// Mitsubishi GX Developer project: 310HGV18J11Y减 改扫码181011   PLC: FX3G

PROGRAM MAIN
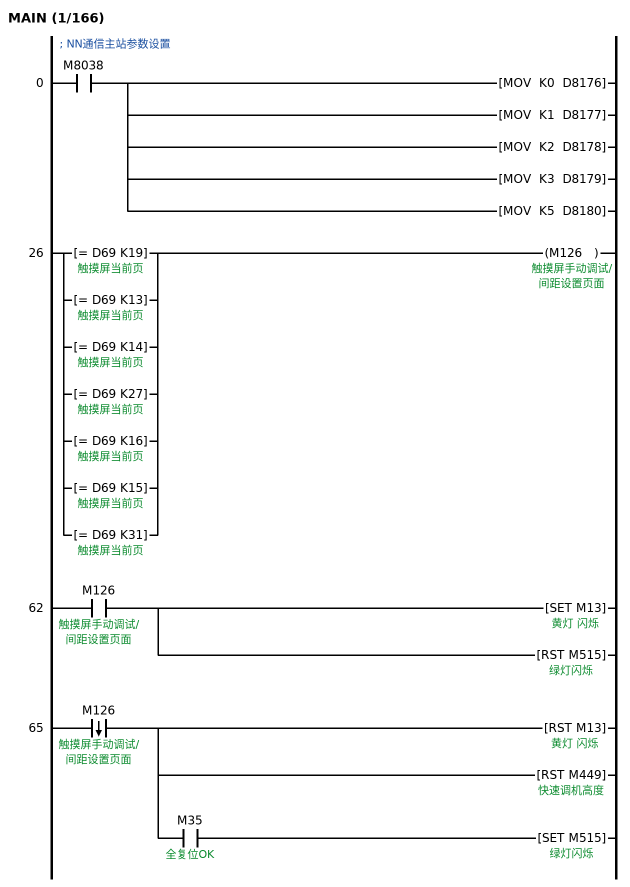
; NN通信主站参数设置
0     LD      M8038
      MOV     K0 D8176
      MOV     K1 D8177
      MOV     K2 D8178
      MOV     K3 D8179
      MOV     K5 D8180
26    LD=     D69 K19  ; 触摸屏当前页
      OR=     D69 K13  ; 触摸屏当前页
      OR=     D69 K14  ; 触摸屏当前页
      OR=     D69 K27  ; 触摸屏当前页
      OR=     D69 K16  ; 触摸屏当前页
      OR=     D69 K15  ; 触摸屏当前页
      OR=     D69 K31  ; 触摸屏当前页
      OUT     M126  ; 触摸屏手动调试/间距设置页面
62    LD      M126  ; 触摸屏手动调试/间距设置页面
      SET     M13  ; 黄灯 闪烁
      RST     M515  ; 绿灯闪烁
65    LDF     M126  ; 触摸屏手动调试/间距设置页面
      RST     M13  ; 黄灯 闪烁
      RST     M449  ; 快速调机高度
      AND     M35  ; 全复位OK
      SET     M515  ; 绿灯闪烁
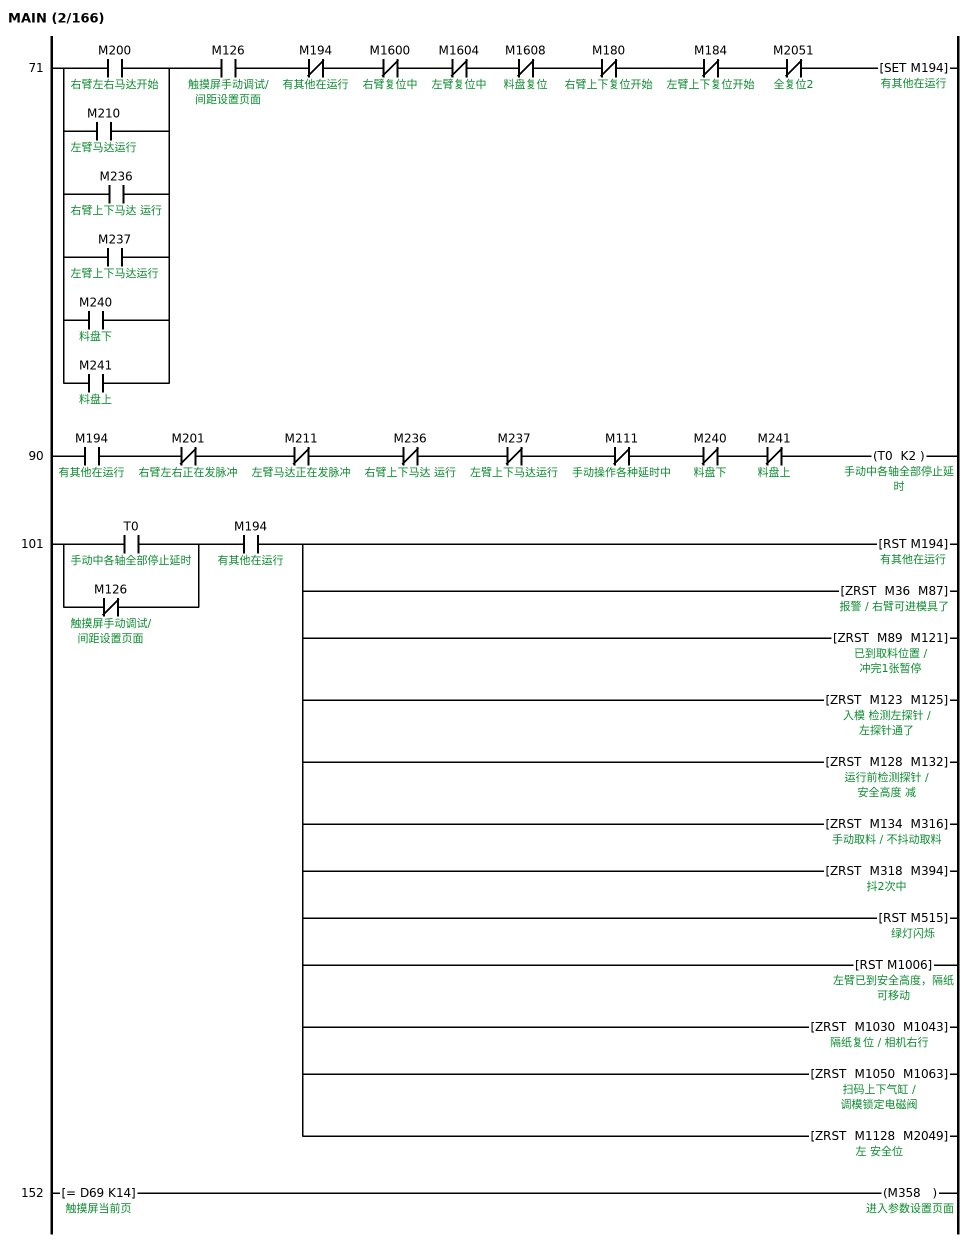
71    LD      M200  ; 右臂左右马达开始
      OR      M210  ; 左臂马达运行
      OR      M236  ; 右臂上下马达 运行
      OR      M237  ; 左臂上下马达运行
      OR      M240  ; 料盘下
      OR      M241  ; 料盘上
      AND     M126  ; 触摸屏手动调试/间距设置页面
      ANI     M194  ; 有其他在运行
      ANI     M1600  ; 右臂复位中
      ANI     M1604  ; 左臂复位中
      ANI     M1608  ; 料盘复位
      ANI     M180  ; 右臂上下复位开始
      ANI     M184  ; 左臂上下复位开始
      ANI     M2051  ; 全复位2
      SET     M194  ; 有其他在运行
90    LD      M194  ; 有其他在运行
      ANI     M201  ; 右臂左右正在发脉冲
      ANI     M211  ; 左臂马达正在发脉冲
      ANI     M236  ; 右臂上下马达 运行
      ANI     M237  ; 左臂上下马达运行
      ANI     M111  ; 手动操作各种延时中
      ANI     M240  ; 料盘下
      ANI     M241  ; 料盘上
      OUT     T0 K2  ; 手动中各轴全部停止延时
101   LD      T0  ; 手动中各轴全部停止延时
      ORI     M126  ; 触摸屏手动调试/间距设置页面
      AND     M194  ; 有其他在运行
      RST     M194  ; 有其他在运行
      ZRST    M36 M87  ; 报警 / 右臂可进模具了
      ZRST    M89 M121  ; 已到取料位置 / 冲完1张暂停
      ZRST    M123 M125  ; 入模 检测左探针 / 左探针通了
      ZRST    M128 M132  ; 运行前检测探针 / 安全高度 减
      ZRST    M134 M316  ; 手动取料 / 不抖动取料
      ZRST    M318 M394  ; 抖2次中
      RST     M515  ; 绿灯闪烁
      RST     M1006  ; 左臂已到安全高度，隔纸可移动
      ZRST    M1030 M1043  ; 隔纸复位 / 相机右行
      ZRST    M1050 M1063  ; 扫码上下气缸 / 调模锁定电磁阀
      ZRST    M1128 M2049  ; 左 安全位
152   LD=     D69 K14  ; 触摸屏当前页
      OUT     M358  ; 进入参数设置页面
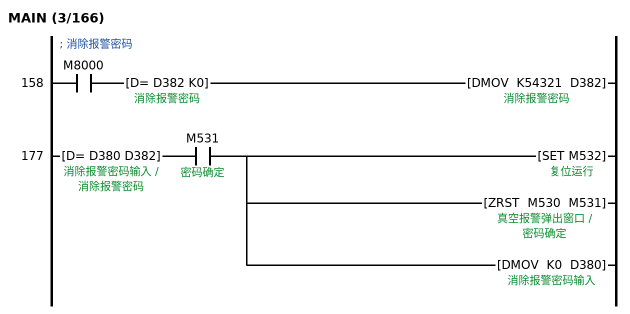
; 消除报警密码
158   LD      M8000
      ANDD=   D382 K0  ; 消除报警密码
      DMOV    K54321 D382
177   LDD=    D380 D382  ; 消除报警密码输入 / 消除报警密码
      AND     M531  ; 密码确定
      SET     M532  ; 复位运行
      ZRST    M530 M531  ; 真空报警弹出窗口
      DMOV    K0 D380
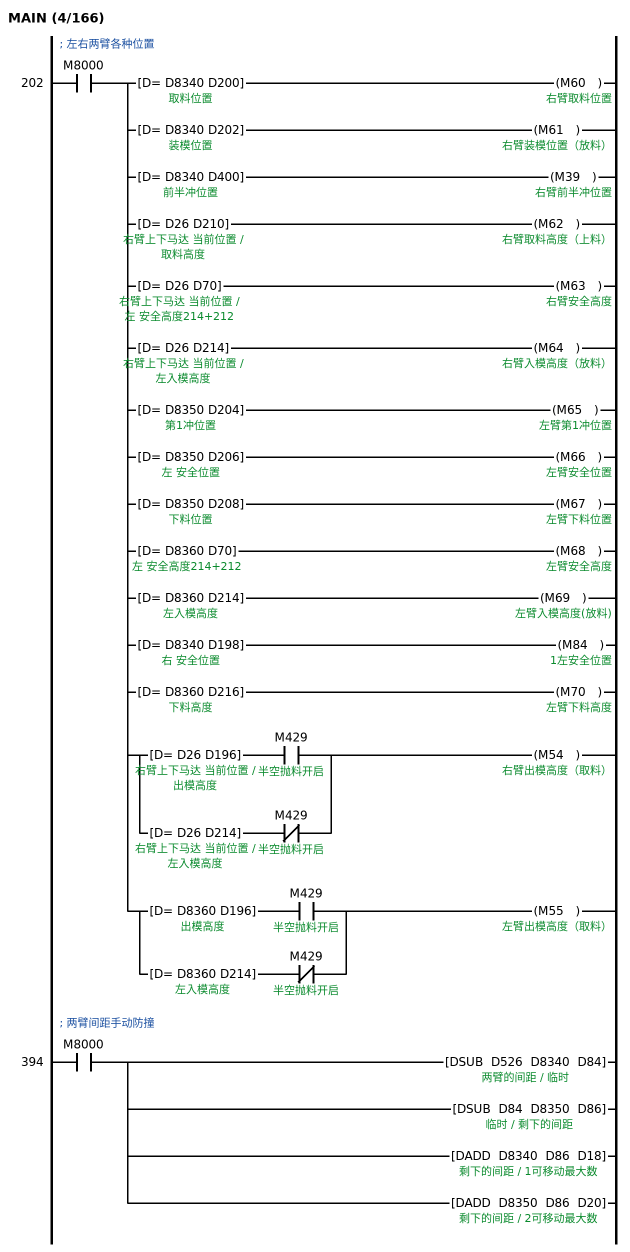
; 左右两臂各种位置
202   LD      M8000
      MPS
      ANDD=   D8340 D200  ; 取料位置
      OUT     M60  ; 右臂取料位置
      MRD
      ANDD=   D8340 D202  ; 装模位置
      OUT     M61  ; 右臂装模位置（放料）
      MRD
      ANDD=   D8340 D400  ; 前半冲位置
      OUT     M39  ; 右臂前半冲位置
      MRD
      ANDD=   D26 D210  ; 右臂上下马达 当前位置 / 取料高度
      OUT     M62  ; 右臂取料高度（上料）
      MRD
      ANDD=   D26 D70  ; 右臂上下马达 当前位置 / 左 安全高度214+212
      OUT     M63  ; 右臂安全高度
      MRD
      ANDD=   D26 D214  ; 右臂上下马达 当前位置 / 左入模高度
      OUT     M64  ; 右臂入模高度（放料）
      MRD
      ANDD=   D8350 D204  ; 第1冲位置
      OUT     M65  ; 左臂第1冲位置
      MRD
      ANDD=   D8350 D206  ; 左 安全位置
      OUT     M66  ; 左臂安全位置
      MRD
      ANDD=   D8350 D208  ; 下料位置
      OUT     M67  ; 左臂下料位置
      MRD
      ANDD=   D8360 D70  ; 左 安全高度214+212
      OUT     M68  ; 左臂安全高度
      MRD
      ANDD=   D8360 D214  ; 左入模高度
      OUT     M69  ; 左臂入模高度(放料)
      MRD
      ANDD=   D8340 D198  ; 右 安全位置
      OUT     M84  ; 1左安全位置
      MRD
      ANDD=   D8360 D216  ; 下料高度
      OUT     M70  ; 左臂下料高度
      MRD
      LDD=    D26 D196  ; 右臂上下马达 当前位置 / 出模高度
      AND     M429  ; 半空抛料开启
      LDD=    D26 D214  ; 右臂上下马达 当前位置 / 左入模高度
      ANI     M429  ; 半空抛料开启
      ORB
      ANB
      OUT     M54  ; 右臂出模高度（取料）
      MPP
      LDD=    D8360 D196  ; 出模高度
      AND     M429  ; 半空抛料开启
      LDD=    D8360 D214  ; 左入模高度
      ANI     M429  ; 半空抛料开启
      ORB
      ANB
      OUT     M55  ; 左臂出模高度（取料）
; 两臂间距手动防撞
394   LD      M8000
      DSUB    D526 D8340 D84  ; 两臂的间距 / 临时
      DSUB    D84 D8350 D86  ; 剩下的间距
      DADD    D8340 D86 D18  ; 1可移动最大数
      DADD    D8350 D86 D20  ; 2可移动最大数
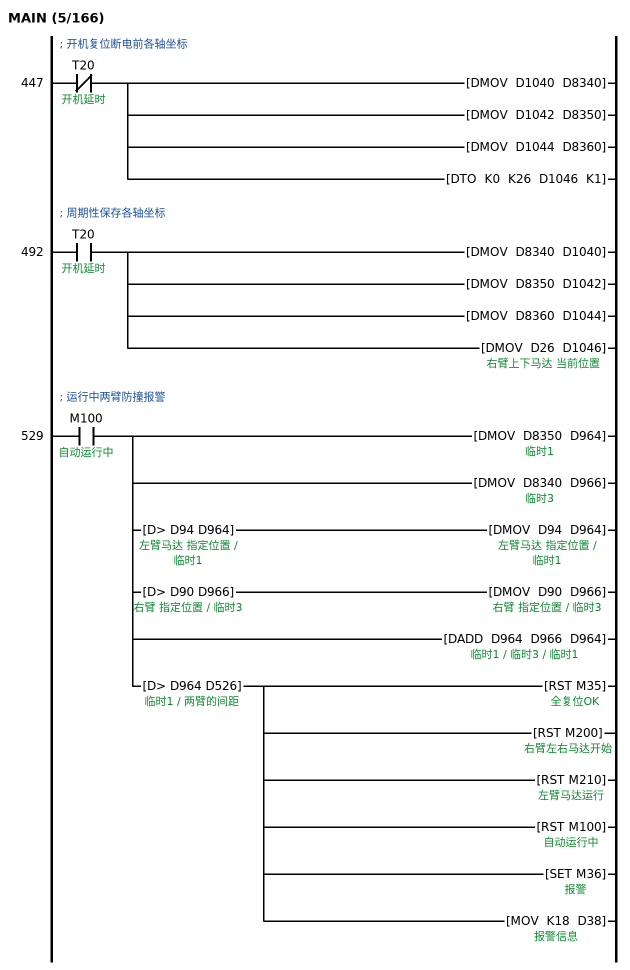
; 开机复位断电前各轴坐标
447   LDI     T20  ; 开机延时
      DMOV    D1040 D8340
      DMOV    D1042 D8350
      DMOV    D1044 D8360
      DTO     K0 K26 D1046 K1
; 周期性保存各轴坐标
492   LD      T20  ; 开机延时
      DMOV    D8340 D1040
      DMOV    D8350 D1042
      DMOV    D8360 D1044
      DMOV    D26 D1046
; 运行中两臂防撞报警
529   LD      M100  ; 自动运行中
      DMOV    D8350 D964  ; 临时1
      DMOV    D8340 D966  ; 临时3
      MPS
      ANDD>   D94 D964  ; 左臂马达 指定位置 / 临时1
      DMOV    D94 D964
      MRD
      ANDD>   D90 D966  ; 右臂 指定位置 / 临时3
      DMOV    D90 D966
      MPP
      DADD    D964 D966 D964
      ANDD>   D964 D526  ; 临时1 / 两臂的间距
      RST     M35  ; 全复位OK
      RST     M200  ; 右臂左右马达开始
      RST     M210  ; 左臂马达运行
      RST     M100  ; 自动运行中
      SET     M36  ; 报警
      MOV     K18 D38  ; 报警信息
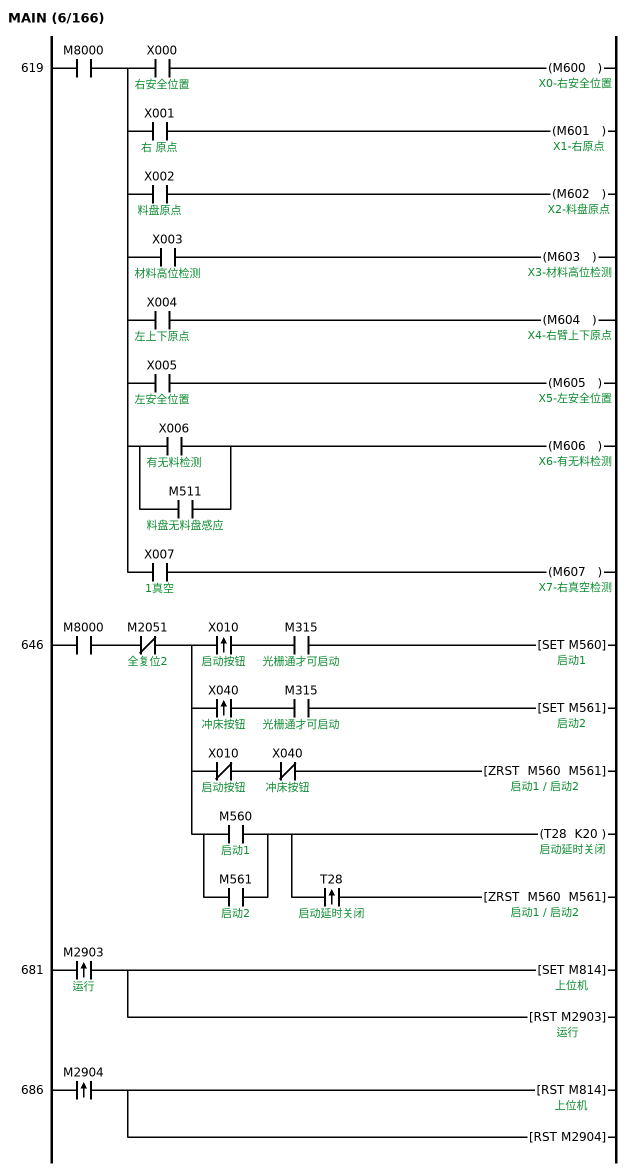
619   LD      M8000
      MPS
      AND     X000  ; 右安全位置
      OUT     M600  ; X0-右安全位置
      MRD
      AND     X001  ; 右 原点
      OUT     M601  ; X1-右原点
      MRD
      AND     X002  ; 料盘原点
      OUT     M602  ; X2-料盘原点
      MRD
      AND     X003  ; 材料高位检测
      OUT     M603  ; X3-材料高位检测
      MRD
      AND     X004  ; 左上下原点
      OUT     M604  ; X4-右臂上下原点
      MRD
      AND     X005  ; 左安全位置
      OUT     M605  ; X5-左安全位置
      MRD
      LD      X006  ; 有无料检测
      OR      M511  ; 料盘无料盘感应
      ANB
      OUT     M606  ; X6-有无料检测
      MPP
      AND     X007  ; 1真空
      OUT     M607  ; X7-右真空检测
646   LD      M8000
      ANI     M2051  ; 全复位2
      MPS
      ANDP    X010  ; 启动按钮
      AND     M315  ; 光栅通才可启动
      SET     M560  ; 启动1
      MRD
      ANDP    X040  ; 冲床按钮
      AND     M315  ; 光栅通才可启动
      SET     M561  ; 启动2
      MRD
      ANI     X010  ; 启动按钮
      ANI     X040  ; 冲床按钮
      ZRST    M560 M561
      MPP
      LD      M560  ; 启动1
      OR      M561  ; 启动2
      ANB
      OUT     T28 K20  ; 启动延时关闭
      ANDP    T28  ; 启动延时关闭
      ZRST    M560 M561
681   LDP     M2903  ; 运行
      SET     M814  ; 上位机
      RST     M2903  ; 运行
686   LDP     M2904
      RST     M814  ; 上位机
      RST     M2904
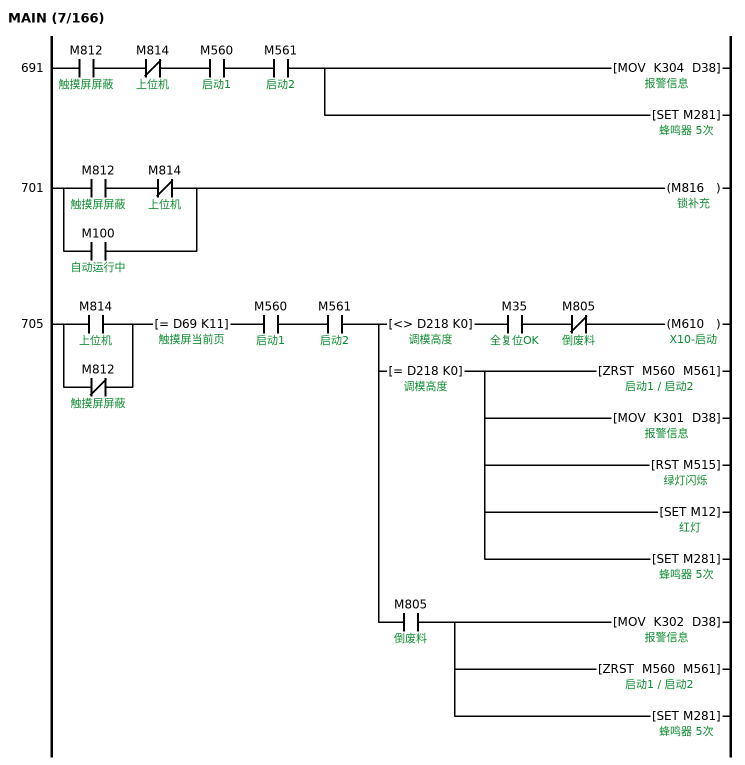
691   LD      M812  ; 触摸屏屏蔽
      ANI     M814  ; 上位机
      AND     M560  ; 启动1
      AND     M561  ; 启动2
      MOV     K304 D38
      SET     M281  ; 蜂鸣器 5次
701   LD      M812  ; 触摸屏屏蔽
      ANI     M814  ; 上位机
      OR      M100  ; 自动运行中
      OUT     M816  ; 锁补充
705   LD      M814  ; 上位机
      ORI     M812  ; 触摸屏屏蔽
      AND=    D69 K11  ; 触摸屏当前页
      AND     M560  ; 启动1
      AND     M561  ; 启动2
      MPS
      AND<>   D218 K0  ; 调模高度
      AND     M35  ; 全复位OK
      ANI     M805  ; 倒废料
      OUT     M610  ; X10-启动
      MRD
      AND=    D218 K0  ; 调模高度
      ZRST    M560 M561
      MOV     K301 D38
      RST     M515  ; 绿灯闪烁
      SET     M12  ; 红灯
      SET     M281  ; 蜂鸣器 5次
      MPP
      AND     M805  ; 倒废料
      MOV     K302 D38
      ZRST    M560 M561
      SET     M281  ; 蜂鸣器 5次
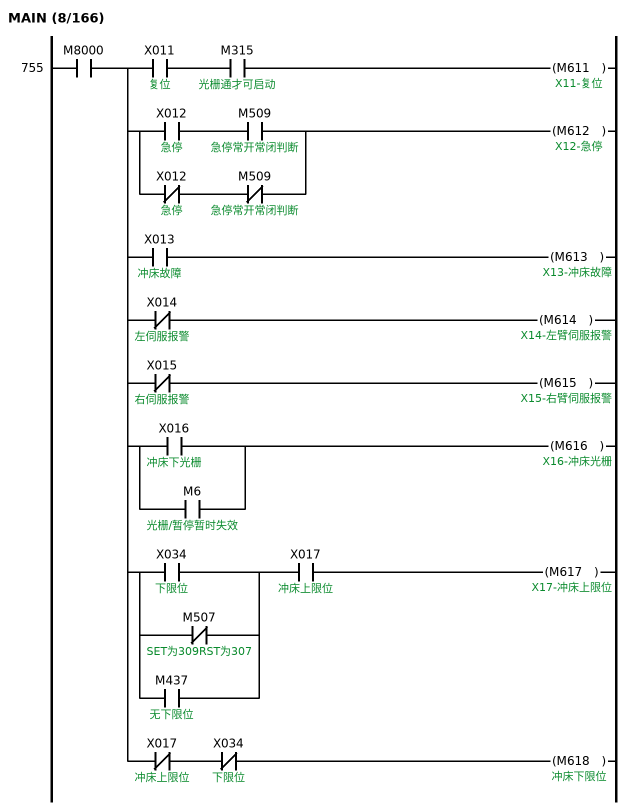
755   LD      M8000
      MPS
      AND     X011  ; 复位
      AND     M315  ; 光栅通才可启动
      OUT     M611  ; X11-复位
      MRD
      LD      X012  ; 急停
      AND     M509  ; 急停常开常闭判断
      LDI     X012  ; 急停
      ANI     M509  ; 急停常开常闭判断
      ORB
      ANB
      OUT     M612  ; X12-急停
      MRD
      AND     X013  ; 冲床故障
      OUT     M613  ; X13-冲床故障
      MRD
      ANI     X014  ; 左伺服报警
      OUT     M614  ; X14-左臂伺服报警
      MRD
      ANI     X015  ; 右伺服报警
      OUT     M615  ; X15-右臂伺服报警
      MRD
      LD      X016  ; 冲床下光栅
      OR      M6  ; 光栅/暂停暂时失效
      ANB
      OUT     M616  ; X16-冲床光栅
      MRD
      LD      X034  ; 下限位
      ORI     M507  ; SET为309RST为307
      OR      M437  ; 无下限位
      ANB
      AND     X017  ; 冲床上限位
      OUT     M617  ; X17-冲床上限位
      MPP
      ANI     X017  ; 冲床上限位
      ANI     X034  ; 下限位
      OUT     M618  ; 冲床下限位
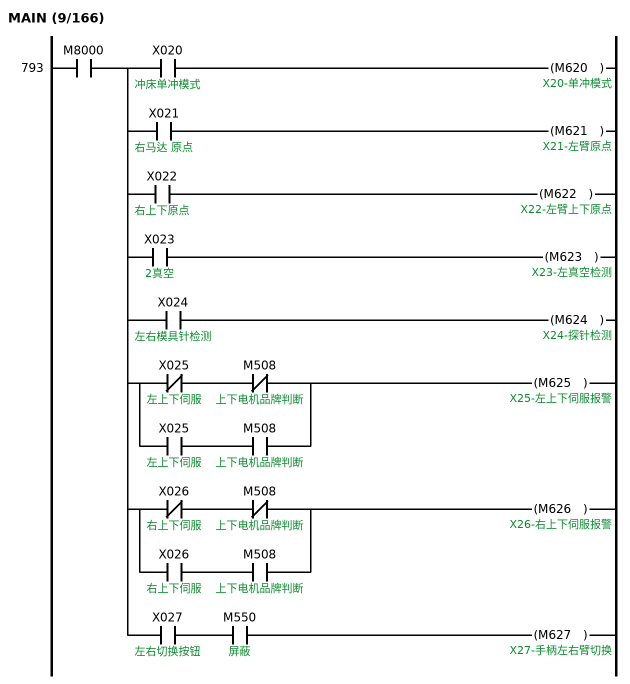
793   LD      M8000
      MPS
      AND     X020  ; 冲床单冲模式
      OUT     M620  ; X20-单冲模式
      MRD
      AND     X021  ; 右马达 原点
      OUT     M621  ; X21-左臂原点
      MRD
      AND     X022  ; 右上下原点
      OUT     M622  ; X22-左臂上下原点
      MRD
      AND     X023  ; 2真空
      OUT     M623  ; X23-左真空检测
      MRD
      AND     X024  ; 左右模具针检测
      OUT     M624  ; X24-探针检测
      MRD
      LDI     X025  ; 左上下伺服
      ANI     M508  ; 上下电机品牌判断
      LD      X025  ; 左上下伺服
      AND     M508  ; 上下电机品牌判断
      ORB
      ANB
      OUT     M625  ; X25-左上下伺服报警
      MRD
      LDI     X026  ; 右上下伺服
      ANI     M508  ; 上下电机品牌判断
      LD      X026  ; 右上下伺服
      AND     M508  ; 上下电机品牌判断
      ORB
      ANB
      OUT     M626  ; X26-右上下伺服报警
      MPP
      AND     X027  ; 左右切换按钮
      AND     M550  ; 屏蔽
      OUT     M627  ; X27-手柄左右臂切换
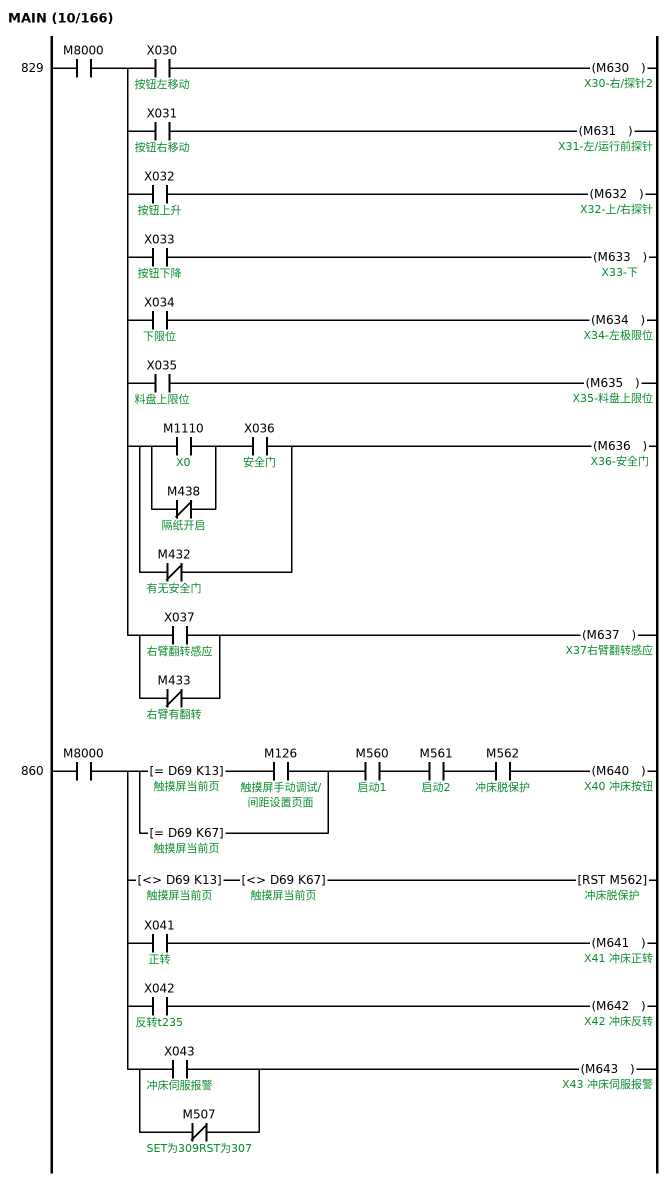
829   LD      M8000
      MPS
      AND     X030  ; 按钮左移动
      OUT     M630  ; X30-右/探针2
      MRD
      AND     X031  ; 按钮右移动
      OUT     M631  ; X31-左/运行前探针
      MRD
      AND     X032  ; 按钮上升
      OUT     M632  ; X32-上/右探针
      MRD
      AND     X033  ; 按钮下降
      OUT     M633  ; X33-下
      MRD
      AND     X034  ; 下限位
      OUT     M634  ; X34-左极限位
      MRD
      AND     X035  ; 料盘上限位
      OUT     M635  ; X35-料盘上限位
      MRD
      LD      M1110  ; X0
      ORI     M438  ; 隔纸开启
      AND     X036  ; 安全门
      ORI     M432  ; 有无安全门
      ANB
      OUT     M636  ; X36-安全门
      MPP
      LD      X037  ; 右臂翻转感应
      ORI     M433  ; 右臂有翻转
      ANB
      OUT     M637  ; X37右臂翻转感应
860   LD      M8000
      MPS
      LD=     D69 K13  ; 触摸屏当前页
      AND     M126  ; 触摸屏手动调试/间距设置页面
      OR=     D69 K67  ; 触摸屏当前页
      ANB
      AND     M560  ; 启动1
      AND     M561  ; 启动2
      AND     M562  ; 冲床脱保护
      OUT     M640  ; X40 冲床按钮
      MRD
      AND<>   D69 K13  ; 触摸屏当前页
      AND<>   D69 K67  ; 触摸屏当前页
      RST     M562  ; 冲床脱保护
      MRD
      AND     X041  ; 正转
      OUT     M641  ; X41 冲床正转
      MRD
      AND     X042  ; 反转t235
      OUT     M642  ; X42 冲床反转
      MPP
      LD      X043  ; 冲床伺服报警
      ORI     M507  ; SET为309RST为307
      ANB
      OUT     M643  ; X43 冲床伺服报警
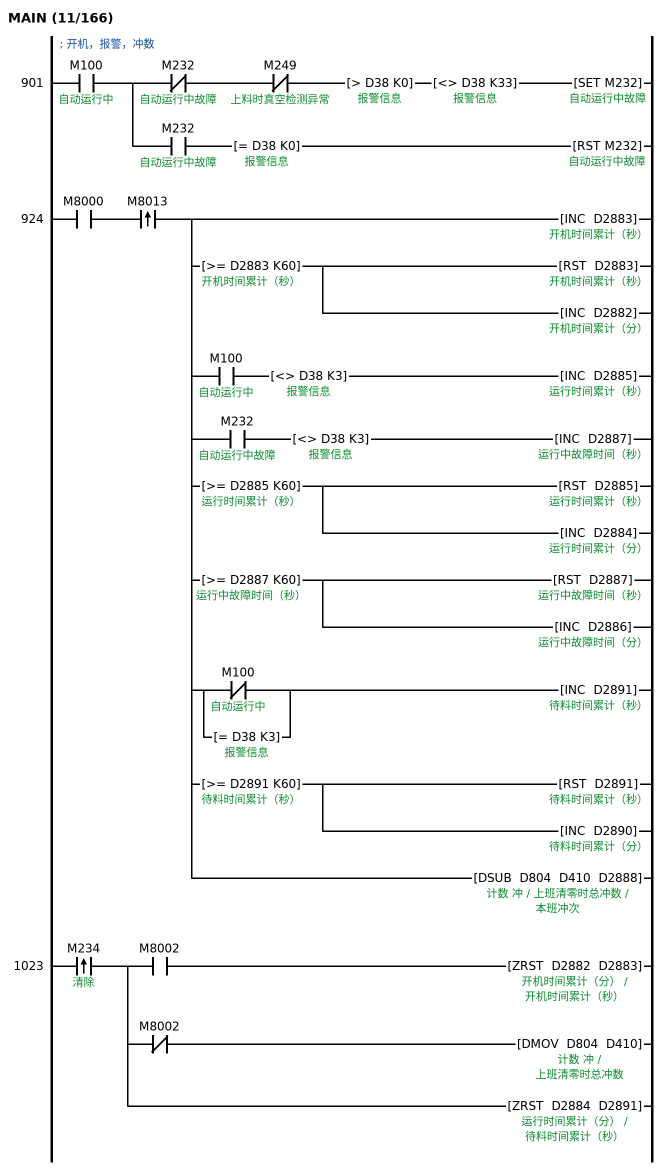
; 开机，报警，冲数
901   LD      M100  ; 自动运行中
      MPS
      ANI     M232  ; 自动运行中故障
      ANI     M249  ; 上料时真空检测异常
      AND>    D38 K0  ; 报警信息
      AND<>   D38 K33  ; 报警信息
      SET     M232  ; 自动运行中故障
      MPP
      AND     M232  ; 自动运行中故障
      AND=    D38 K0  ; 报警信息
      RST     M232  ; 自动运行中故障
924   LD      M8000
      ANDP    M8013
      INC     D2883  ; 开机时间累计（秒）
      MPS
      AND>=   D2883 K60  ; 开机时间累计（秒）
      RST     D2883  ; 开机时间累计（秒）
      INC     D2882  ; 开机时间累计（分）
      MRD
      AND     M100  ; 自动运行中
      AND<>   D38 K3  ; 报警信息
      INC     D2885  ; 运行时间累计（秒）
      MRD
      AND     M232  ; 自动运行中故障
      AND<>   D38 K3  ; 报警信息
      INC     D2887  ; 运行中故障时间（秒）
      MRD
      AND>=   D2885 K60  ; 运行时间累计（秒）
      RST     D2885  ; 运行时间累计（秒）
      INC     D2884  ; 运行时间累计（分）
      MRD
      AND>=   D2887 K60  ; 运行中故障时间（秒）
      RST     D2887  ; 运行中故障时间（秒）
      INC     D2886  ; 运行中故障时间（分）
      MRD
      LDI     M100  ; 自动运行中
      OR=     D38 K3  ; 报警信息
      ANB
      INC     D2891  ; 待料时间累计（秒）
      MRD
      AND>=   D2891 K60  ; 待料时间累计（秒）
      RST     D2891  ; 待料时间累计（秒）
      INC     D2890  ; 待料时间累计（分）
      MPP
      DSUB    D804 D410 D2888  ; 计数 冲 / 上班清零时总冲数 / 本班冲次
1023  LDP     M234  ; 清除
      MPS
      AND     M8002
      ZRST    D2882 D2883
      MRD
      ANI     M8002
      DMOV    D804 D410
      MPP
      ZRST    D2884 D2891
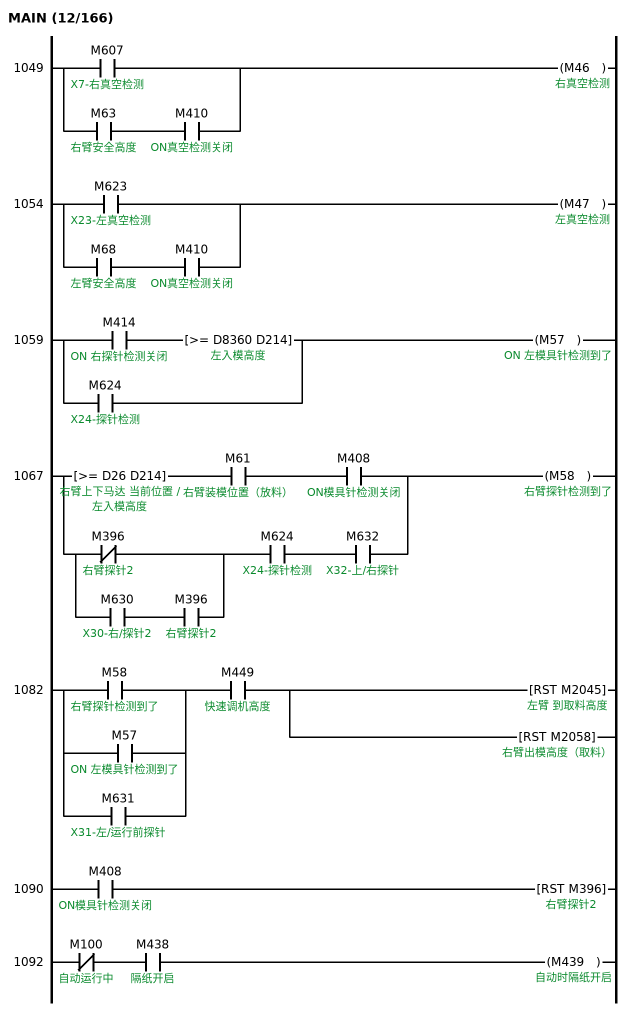
1049  LD      M607  ; X7-右真空检测
      LD      M63  ; 右臂安全高度
      AND     M410  ; ON真空检测关闭
      ORB
      OUT     M46  ; 右真空检测
1054  LD      M623  ; X23-左真空检测
      LD      M68  ; 左臂安全高度
      AND     M410  ; ON真空检测关闭
      ORB
      OUT     M47  ; 左真空检测
1059  LD      M414  ; ON 右探针检测关闭
      AND>=   D8360 D214  ; 左入模高度
      OR      M624  ; X24-探针检测
      OUT     M57  ; ON 左模具针检测到了
1067  LD>=    D26 D214  ; 右臂上下马达 当前位置 / 左入模高度
      AND     M61  ; 右臂装模位置（放料）
      AND     M408  ; ON模具针检测关闭
      LDI     M396  ; 右臂探针2
      LD      M630  ; X30-右/探针2
      AND     M396  ; 右臂探针2
      ORB
      AND     M624  ; X24-探针检测
      AND     M632  ; X32-上/右探针
      ORB
      OUT     M58  ; 右臂探针检测到了
1082  LD      M58  ; 右臂探针检测到了
      OR      M57  ; ON 左模具针检测到了
      OR      M631  ; X31-左/运行前探针
      AND     M449  ; 快速调机高度
      RST     M2045  ; 左臂 到取料高度
      RST     M2058  ; 右臂出模高度（取料）
1090  LD      M408  ; ON模具针检测关闭
      RST     M396  ; 右臂探针2
1092  LDI     M100  ; 自动运行中
      AND     M438  ; 隔纸开启
      OUT     M439  ; 自动时隔纸开启
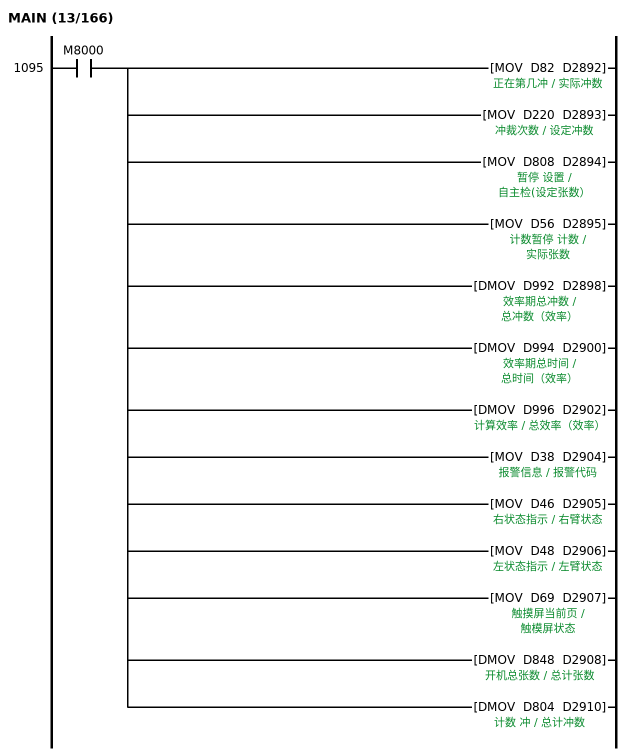
1095  LD      M8000
      MOV     D82 D2892  ; 正在第几冲 / 实际冲数
      MOV     D220 D2893  ; 冲裁次数 / 设定冲数
      MOV     D808 D2894  ; 暂停 设置 / 自主检(设定张数）
      MOV     D56 D2895  ; 计数暂停 计数 / 实际张数
      DMOV    D992 D2898  ; 效率期总冲数 / 总冲数（效率）
      DMOV    D994 D2900  ; 效率期总时间 / 总时间（效率）
      DMOV    D996 D2902  ; 计算效率 / 总效率（效率）
      MOV     D38 D2904  ; 报警代码
      MOV     D46 D2905  ; 右状态指示 / 右臂状态
      MOV     D48 D2906  ; 左状态指示 / 左臂状态
      MOV     D69 D2907  ; 触模屏状态
      DMOV    D848 D2908  ; 开机总张数 / 总计张数
      DMOV    D804 D2910  ; 总计冲数
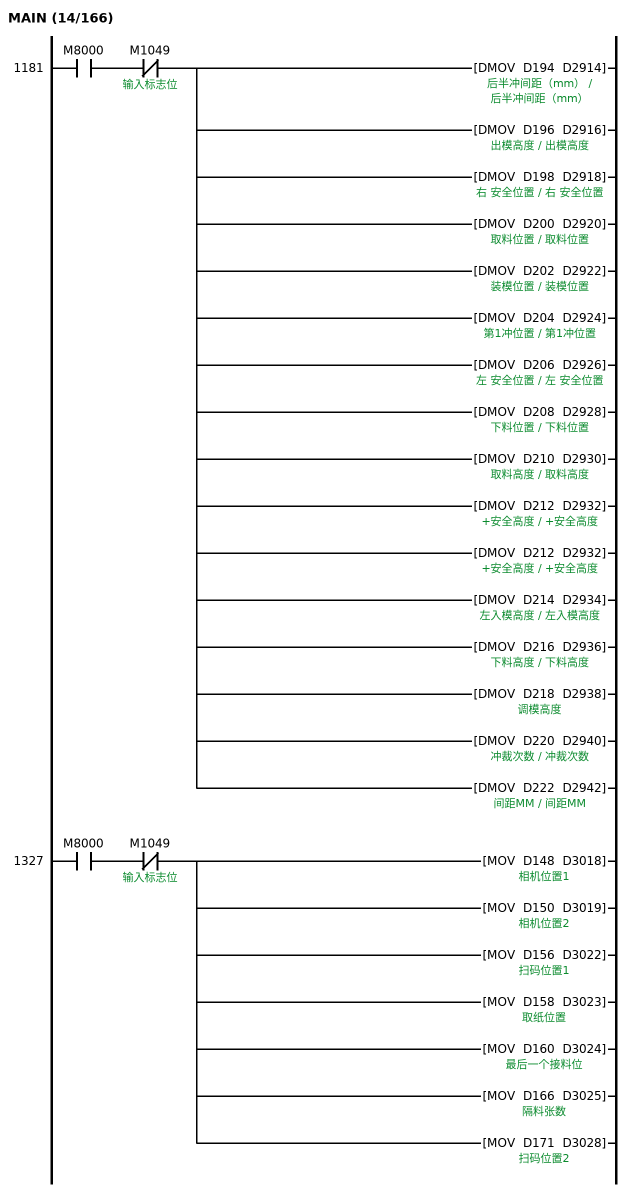
1181  LD      M8000
      ANI     M1049  ; 输入标志位
      DMOV    D194 D2914  ; 后半冲间距（mm） / 后半冲间距（mm）
      DMOV    D196 D2916  ; 出模高度
      DMOV    D198 D2918  ; 右 安全位置
      DMOV    D200 D2920  ; 取料位置
      DMOV    D202 D2922  ; 装模位置
      DMOV    D204 D2924  ; 第1冲位置
      DMOV    D206 D2926  ; 左 安全位置
      DMOV    D208 D2928  ; 下料位置
      DMOV    D210 D2930  ; 取料高度
      DMOV    D212 D2932  ; +安全高度 / +安全高度
      DMOV    D212 D2932
      DMOV    D214 D2934  ; 左入模高度
      DMOV    D216 D2936  ; 下料高度
      DMOV    D218 D2938
      DMOV    D220 D2940  ; 冲裁次数
      DMOV    D222 D2942  ; 间距MM / 间距MM
1327  LD      M8000
      ANI     M1049  ; 输入标志位
      MOV     D148 D3018  ; 相机位置1
      MOV     D150 D3019  ; 相机位置2
      MOV     D156 D3022  ; 扫码位置1
      MOV     D158 D3023  ; 取纸位置
      MOV     D160 D3024  ; 最后一个接料位
      MOV     D166 D3025  ; 隔料张数
      MOV     D171 D3028  ; 扫码位置2
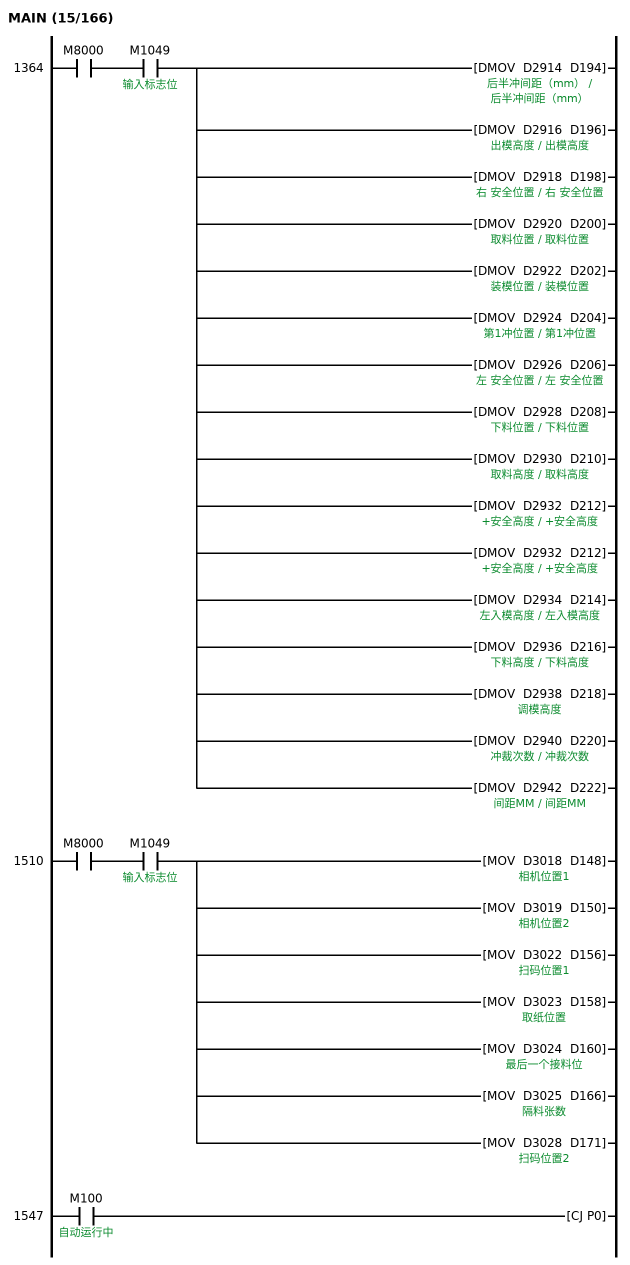
1364  LD      M8000
      AND     M1049  ; 输入标志位
      DMOV    D2914 D194
      DMOV    D2916 D196
      DMOV    D2918 D198
      DMOV    D2920 D200
      DMOV    D2922 D202
      DMOV    D2924 D204
      DMOV    D2926 D206
      DMOV    D2928 D208
      DMOV    D2930 D210
      DMOV    D2932 D212
      DMOV    D2932 D212
      DMOV    D2934 D214
      DMOV    D2936 D216
      DMOV    D2938 D218
      DMOV    D2940 D220
      DMOV    D2942 D222
1510  LD      M8000
      AND     M1049  ; 输入标志位
      MOV     D3018 D148
      MOV     D3019 D150
      MOV     D3022 D156
      MOV     D3023 D158
      MOV     D3024 D160
      MOV     D3025 D166
      MOV     D3028 D171
1547  LD      M100  ; 自动运行中
      CJ      P0
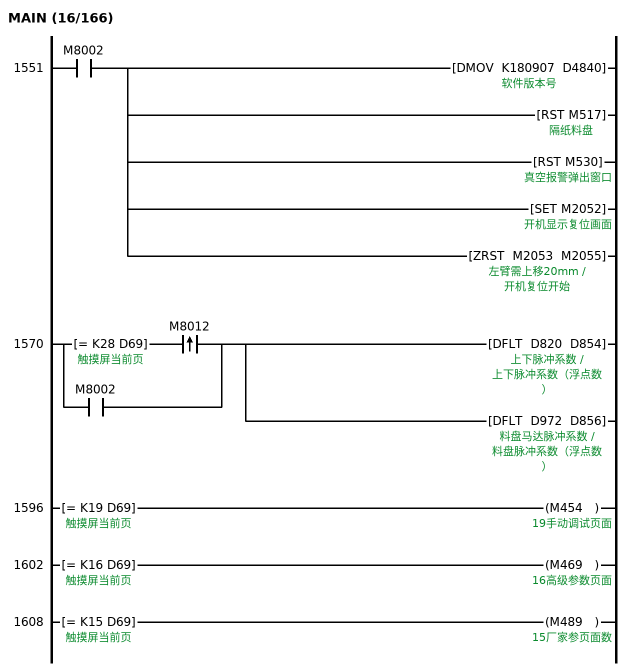
1551  LD      M8002
      DMOV    K180907 D4840  ; 软件版本号
      RST     M517  ; 隔纸料盘
      RST     M530  ; 真空报警弹出窗口
      SET     M2052  ; 开机显示复位画面
      ZRST    M2053 M2055  ; 左臂需上移20mm / 开机复位开始
1570  LD=     K28 D69  ; 触摸屏当前页
      ANDP    M8012
      OR      M8002
      DFLT    D820 D854  ; 上下脉冲系数 / 上下脉冲系数（浮点数）
      DFLT    D972 D856  ; 料盘马达脉冲系数 / 料盘脉冲系数（浮点数）
1596  LD=     K19 D69  ; 触摸屏当前页
      OUT     M454  ; 19手动调试页面
1602  LD=     K16 D69  ; 触摸屏当前页
      OUT     M469  ; 16高级参数页面
1608  LD=     K15 D69  ; 触摸屏当前页
      OUT     M489  ; 15厂家参页面数
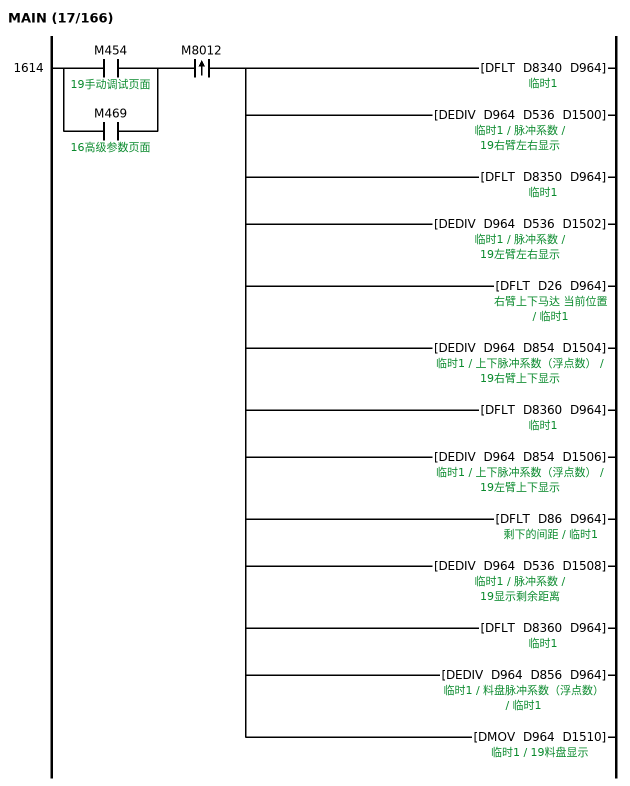
1614  LD      M454  ; 19手动调试页面
      OR      M469  ; 16高级参数页面
      ANDP    M8012
      DFLT    D8340 D964
      DEDIV   D964 D536 D1500  ; 脉冲系数 / 19右臂左右显示
      DFLT    D8350 D964
      DEDIV   D964 D536 D1502  ; 19左臂左右显示
      DFLT    D26 D964
      DEDIV   D964 D854 D1504  ; 19右臂上下显示
      DFLT    D8360 D964
      DEDIV   D964 D854 D1506  ; 19左臂上下显示
      DFLT    D86 D964
      DEDIV   D964 D536 D1508  ; 19显示剩余距离
      DFLT    D8360 D964
      DEDIV   D964 D856 D964
      DMOV    D964 D1510  ; 19料盘显示
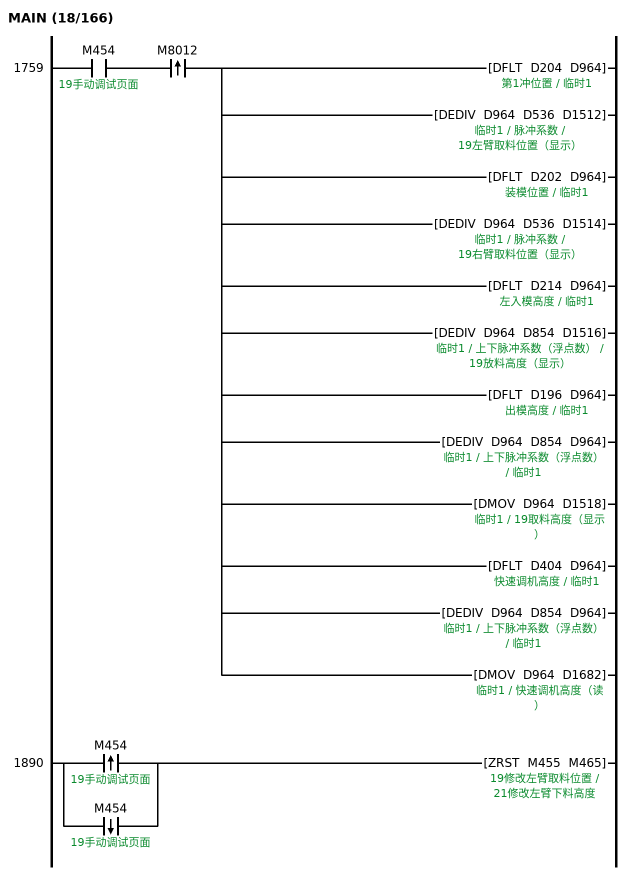
1759  LD      M454  ; 19手动调试页面
      ANDP    M8012
      DFLT    D204 D964
      DEDIV   D964 D536 D1512  ; 19左臂取料位置（显示）
      DFLT    D202 D964
      DEDIV   D964 D536 D1514  ; 19右臂取料位置（显示）
      DFLT    D214 D964
      DEDIV   D964 D854 D1516  ; 19放料高度（显示）
      DFLT    D196 D964
      DEDIV   D964 D854 D964
      DMOV    D964 D1518  ; 19取料高度（显示）
      DFLT    D404 D964  ; 快速调机高度
      DEDIV   D964 D854 D964
      DMOV    D964 D1682  ; 快速调机高度（读）
1890  LDP     M454  ; 19手动调试页面
      ORF     M454  ; 19手动调试页面
      ZRST    M455 M465  ; 19修改左臂取料位置 / 21修改左臂下料高度
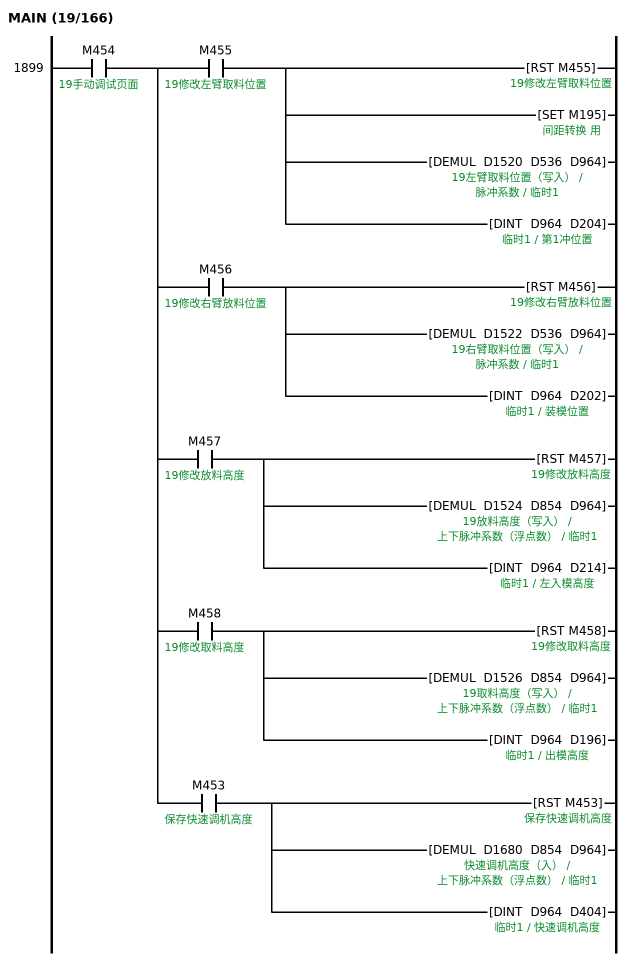
1899  LD      M454  ; 19手动调试页面
      MPS
      AND     M455  ; 19修改左臂取料位置
      RST     M455  ; 19修改左臂取料位置
      SET     M195  ; 间距转换 用
      DEMUL   D1520 D536 D964  ; 19左臂取料位置（写入）
      DINT    D964 D204
      MRD
      AND     M456  ; 19修改右臂放料位置
      RST     M456  ; 19修改右臂放料位置
      DEMUL   D1522 D536 D964  ; 19右臂取料位置（写入）
      DINT    D964 D202
      MRD
      AND     M457  ; 19修改放料高度
      RST     M457  ; 19修改放料高度
      DEMUL   D1524 D854 D964  ; 19放料高度（写入）
      DINT    D964 D214
      MRD
      AND     M458  ; 19修改取料高度
      RST     M458  ; 19修改取料高度
      DEMUL   D1526 D854 D964  ; 19取料高度（写入）
      DINT    D964 D196
      MPP
      AND     M453  ; 保存快速调机高度
      RST     M453  ; 保存快速调机高度
      DEMUL   D1680 D854 D964  ; 快速调机高度（入）
      DINT    D964 D404
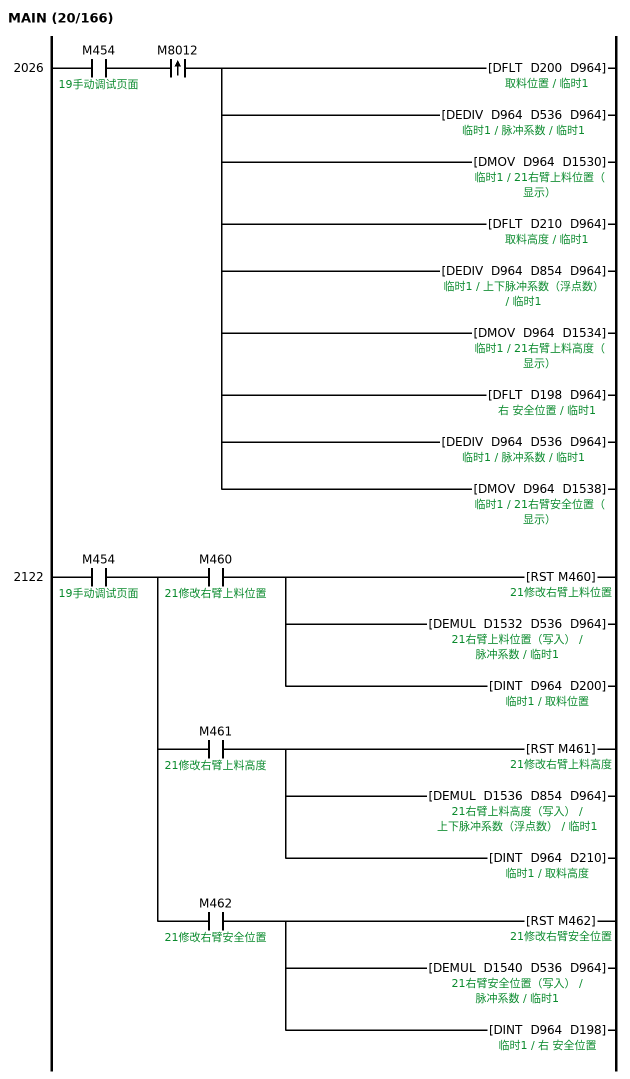
2026  LD      M454  ; 19手动调试页面
      ANDP    M8012
      DFLT    D200 D964
      DEDIV   D964 D536 D964
      DMOV    D964 D1530  ; 21右臂上料位置（显示）
      DFLT    D210 D964
      DEDIV   D964 D854 D964
      DMOV    D964 D1534  ; 21右臂上料高度（显示）
      DFLT    D198 D964
      DEDIV   D964 D536 D964
      DMOV    D964 D1538  ; 21右臂安全位置（显示）
2122  LD      M454  ; 19手动调试页面
      MPS
      AND     M460  ; 21修改右臂上料位置
      RST     M460  ; 21修改右臂上料位置
      DEMUL   D1532 D536 D964  ; 21右臂上料位置（写入）
      DINT    D964 D200
      MRD
      AND     M461  ; 21修改右臂上料高度
      RST     M461  ; 21修改右臂上料高度
      DEMUL   D1536 D854 D964  ; 21右臂上料高度（写入）
      DINT    D964 D210
      MPP
      AND     M462  ; 21修改右臂安全位置
      RST     M462  ; 21修改右臂安全位置
      DEMUL   D1540 D536 D964  ; 21右臂安全位置（写入）
      DINT    D964 D198
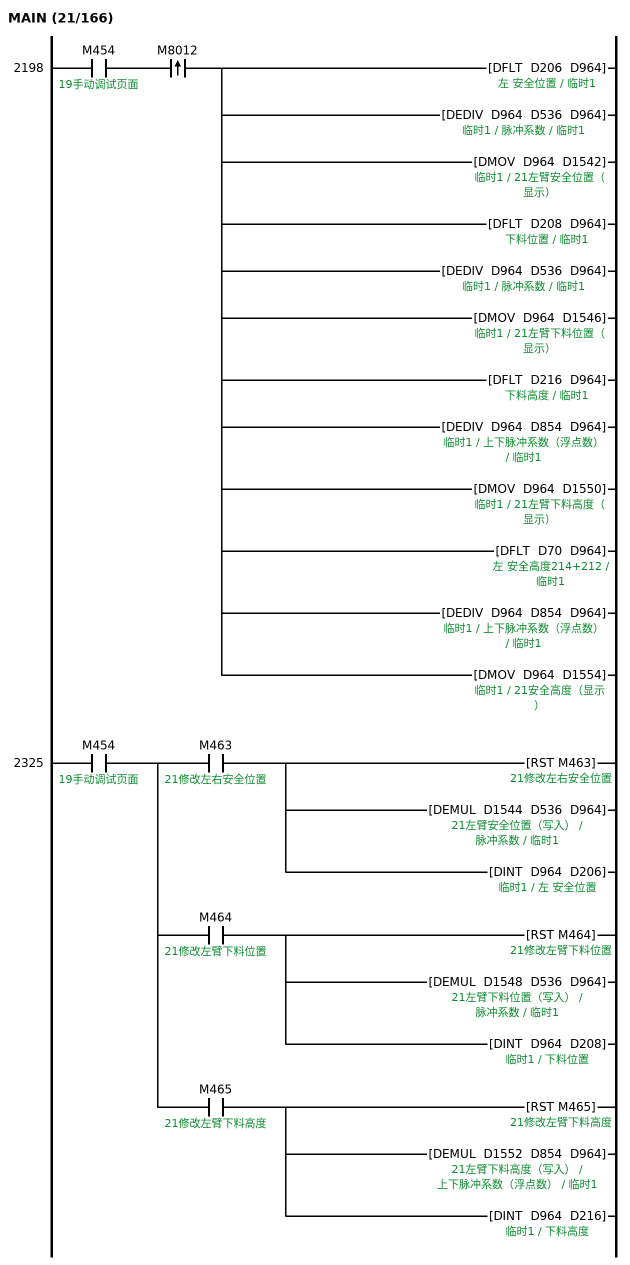
2198  LD      M454  ; 19手动调试页面
      ANDP    M8012
      DFLT    D206 D964
      DEDIV   D964 D536 D964
      DMOV    D964 D1542  ; 21左臂安全位置（显示）
      DFLT    D208 D964
      DEDIV   D964 D536 D964
      DMOV    D964 D1546  ; 21左臂下料位置（显示）
      DFLT    D216 D964
      DEDIV   D964 D854 D964
      DMOV    D964 D1550  ; 21左臂下料高度（显示）
      DFLT    D70 D964
      DEDIV   D964 D854 D964
      DMOV    D964 D1554  ; 21安全高度（显示）
2325  LD      M454  ; 19手动调试页面
      MPS
      AND     M463  ; 21修改左右安全位置
      RST     M463  ; 21修改左右安全位置
      DEMUL   D1544 D536 D964  ; 21左臂安全位置（写入）
      DINT    D964 D206
      MRD
      AND     M464  ; 21修改左臂下料位置
      RST     M464  ; 21修改左臂下料位置
      DEMUL   D1548 D536 D964  ; 21左臂下料位置（写入）
      DINT    D964 D208
      MPP
      AND     M465  ; 21修改左臂下料高度
      RST     M465  ; 21修改左臂下料高度
      DEMUL   D1552 D854 D964  ; 21左臂下料高度（写入）
      DINT    D964 D216
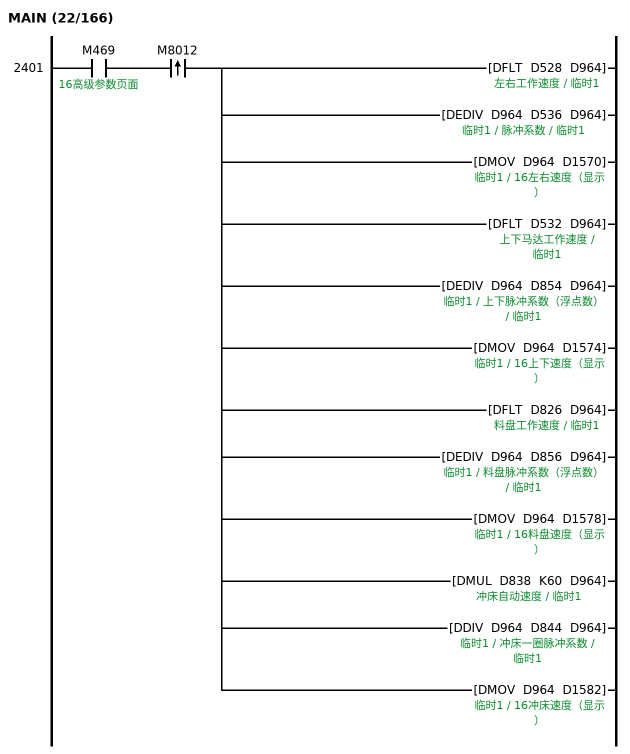
2401  LD      M469  ; 16高级参数页面
      ANDP    M8012
      DFLT    D528 D964  ; 左右工作速度
      DEDIV   D964 D536 D964
      DMOV    D964 D1570  ; 16左右速度（显示）
      DFLT    D532 D964  ; 上下马达工作速度
      DEDIV   D964 D854 D964
      DMOV    D964 D1574  ; 16上下速度（显示）
      DFLT    D826 D964  ; 料盘工作速度
      DEDIV   D964 D856 D964
      DMOV    D964 D1578  ; 16料盘速度（显示）
      DMUL    D838 K60 D964  ; 冲床自动速度
      DDIV    D964 D844 D964  ; 冲床一圈脉冲系数
      DMOV    D964 D1582  ; 16冲床速度（显示）
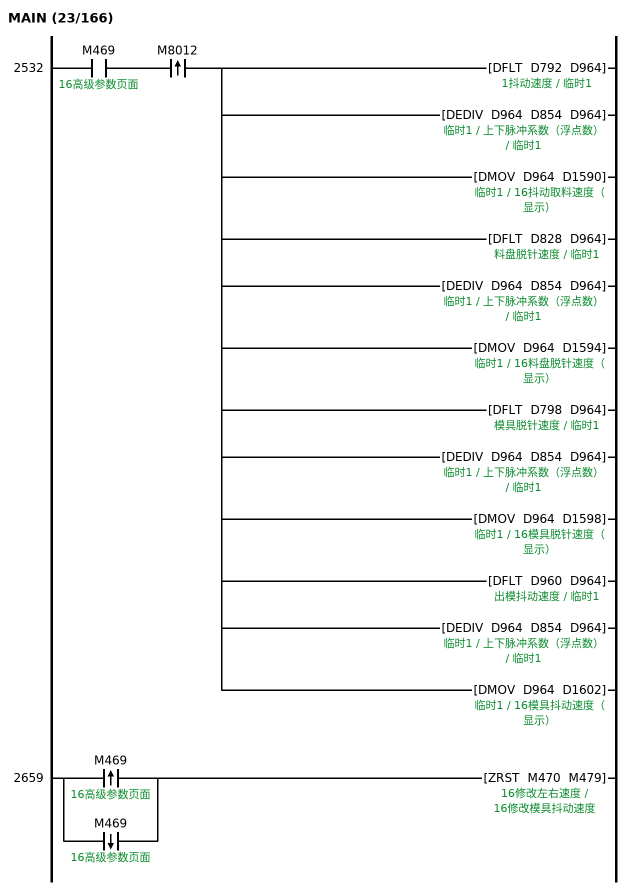
2532  LD      M469  ; 16高级参数页面
      ANDP    M8012
      DFLT    D792 D964  ; 1抖动速度
      DEDIV   D964 D854 D964
      DMOV    D964 D1590  ; 16抖动取料速度（显示）
      DFLT    D828 D964  ; 料盘脱针速度
      DEDIV   D964 D854 D964
      DMOV    D964 D1594  ; 16料盘脱针速度（显示）
      DFLT    D798 D964  ; 模具脱针速度
      DEDIV   D964 D854 D964
      DMOV    D964 D1598  ; 16模具脱针速度（显示）
      DFLT    D960 D964  ; 出模抖动速度
      DEDIV   D964 D854 D964
      DMOV    D964 D1602  ; 16模具抖动速度（显示）
2659  LDP     M469  ; 16高级参数页面
      ORF     M469  ; 16高级参数页面
      ZRST    M470 M479  ; 16修改左右速度 / 16修改模具抖动速度
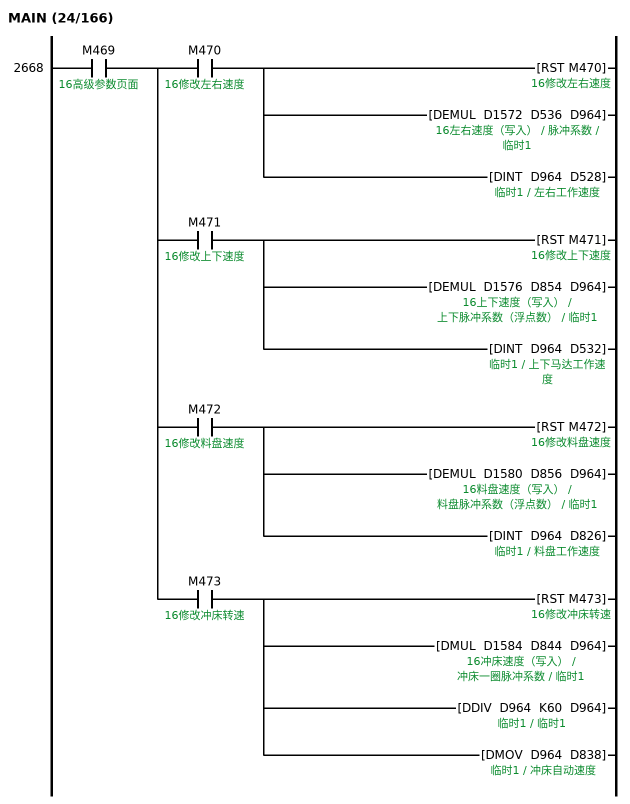
2668  LD      M469  ; 16高级参数页面
      MPS
      AND     M470  ; 16修改左右速度
      RST     M470  ; 16修改左右速度
      DEMUL   D1572 D536 D964  ; 16左右速度（写入）
      DINT    D964 D528
      MRD
      AND     M471  ; 16修改上下速度
      RST     M471  ; 16修改上下速度
      DEMUL   D1576 D854 D964  ; 16上下速度（写入）
      DINT    D964 D532
      MRD
      AND     M472  ; 16修改料盘速度
      RST     M472  ; 16修改料盘速度
      DEMUL   D1580 D856 D964  ; 16料盘速度（写入）
      DINT    D964 D826
      MPP
      AND     M473  ; 16修改冲床转速
      RST     M473  ; 16修改冲床转速
      DMUL    D1584 D844 D964  ; 16冲床速度（写入）
      DDIV    D964 K60 D964
      DMOV    D964 D838
